# EPICS substitutions: blenApp/Db/common/coefTf.substitutions
#scaling for coefficent B and E to account to ln being applied

file coefTransform.db
{
pattern {P, AMC, COEF}

    {$(P), 0, B}
    {$(P), 0, E}
    {$(P), 1, B}
    {$(P), 1, E}
}
